{attribute 'GeneratedUsingTerminal: EPP1342-0001-0016'}
{attribute addProperty BoxType "EPP1342-0001-0016"}
{attribute addProperty Description "EPP1342-0001 3 port EtherCAT P junction"}
{attribute addProperty Physics "YYYY"}
{attribute addProperty Id "InfoDataAT %I*InfoData_6F19DB2B2"}
{attribute addProperty CRC "532711307"}
{attribute addProperty Size "2"}
TYPE EPP1342_1FC0878B EXTENDS EtcSlaveBoxBase_77A0E4A7 :
STRUCT
	{attribute addProperty Name "InfoData"}
	InfoData : InfoData_6F19DB2B;
END_STRUCT
END_TYPE

(* stored: Version 1.2.0.0, ProductVersion 3.1.4024.9
   DUT EPP1342_1FC0878B: Id {68586fab-74a4-425a-82f1-856216ca1bd2} *)
